{attribute 'GeneratedUsingTerminal: EK1122-0000-0018'}
{attribute addProperty BoxType "EK1122-0000-0018"}
{attribute addProperty Id "Beckhoff_EPP3xxxsub_EK1100EK1100_1FC0878B2A_0001_EPP3174_0002_0016EPP3174_DCC7866252A_0002_EPP3174_0002_0017EPP3174_DCC7866252A_0003_EPP3174_0002_0018EPP3174_DCC7866252A_0004_EPP3184_0002_0016EPP3184_DCC7866252A_0005_EPP3184_0002_0017EPP3184_DCC7866252A_0006_EPP3184_0002_0018EPP3184_DCC7866252A_0007_EPP3184_0002_0019EPP3184_DCC7866252A_0008_EPP3204_0002_0016EPP3204_6CD7E11952A_0009_EPP3204_0002_0017EPP3204_5380707048A_0010_EPP3204_0002_0018EPP3204_5380707048A_0011_EPP3204_0002_0019EPP3204_5380707048A_0012_EPP3314_0002_0016EPP3314_B654D23048A_0013_EPP3314_0002_0017EPP3314_B654D23048A_0014_EPP3314_0002_0018EPP3314_B654D23048A_0015_EPP3632_0001_0016EPP3632_E2B98A5C86A_0016_EPP3632_0001_0017EPP3632_E2B98A5C86A_0017_EPP3744_0041_0016EPP3744_315C92D470A_0018_EPP3744_0041_0017EPP3744_315C92D470A_0019_EPP3744_0041_0018EPP3744_315C92D470A_0020_EPP3744_1041_0016EPP3744_315C92D470A_0021_EPP3744_1041_0017EPP3744_315C92D470A_0022_EPP3744_1041_0018EPP3744_315C92D470A_0023_EPP3744_1041_0019EPP3744_315C92D470A_0024_EPP3744_1041_0020EPP3744_315C92D470A_0025_EPP3752_0000_0017EPP3752_C992DA1B42"}
{attribute addProperty CRC "2576063294"}
{attribute addProperty Size "1480"}
TYPE Beckhoff_EPP3xxxEK1122_998B9B3E EXTENDS EK1122_1FC0878B :
STRUCT
	{attribute addProperty Name "Beckhoff_EPP3xxxsub_EK1100"}
	{attribute addProperty PreviousPort "Beckhoff EPP3xxxEK1122 : D"}
	Beckhoff_EPP3xxxsub_EK1100 : EK1100_1FC0878B;
	{attribute addProperty Name "A_0001_EPP3174_0002_0016"}
	{attribute addProperty PreviousPort "Beckhoff EPP3xxxsub EK1100 : C"}
	A_0001_EPP3174_0002_0016 : EPP3174_DCC78662;
	{attribute addProperty Name "A_0002_EPP3174_0002_0017"}
	{attribute addProperty PreviousPort "A_0001(EPP3174-0002-0016) : B"}
	A_0002_EPP3174_0002_0017 : EPP3174_DCC78662;
	{attribute addProperty Name "A_0003_EPP3174_0002_0018"}
	{attribute addProperty PreviousPort "A_0002(EPP3174-0002-0017) : B"}
	A_0003_EPP3174_0002_0018 : EPP3174_DCC78662;
	{attribute addProperty Name "A_0004_EPP3184_0002_0016"}
	{attribute addProperty PreviousPort "A_0003(EPP3174-0002-0018) : B"}
	A_0004_EPP3184_0002_0016 : EPP3184_DCC78662;
	{attribute addProperty Name "A_0005_EPP3184_0002_0017"}
	{attribute addProperty PreviousPort "A_0004(EPP3184-0002-0016) : B"}
	A_0005_EPP3184_0002_0017 : EPP3184_DCC78662;
	{attribute addProperty Name "A_0006_EPP3184_0002_0018"}
	{attribute addProperty PreviousPort "A_0005(EPP3184-0002-0017) : B"}
	A_0006_EPP3184_0002_0018 : EPP3184_DCC78662;
	{attribute addProperty Name "A_0007_EPP3184_0002_0019"}
	{attribute addProperty PreviousPort "A_0006(EPP3184-0002-0018) : B"}
	A_0007_EPP3184_0002_0019 : EPP3184_DCC78662;
	{attribute addProperty Name "A_0008_EPP3204_0002_0016"}
	{attribute addProperty PreviousPort "A_0007(EPP3184-0002-0019) : B"}
	A_0008_EPP3204_0002_0016 : EPP3204_6CD7E119;
	{attribute addProperty Name "A_0009_EPP3204_0002_0017"}
	{attribute addProperty PreviousPort "A_0008(EPP3204-0002-0016) : B"}
	A_0009_EPP3204_0002_0017 : EPP3204_53807070;
	{attribute addProperty Name "A_0010_EPP3204_0002_0018"}
	{attribute addProperty PreviousPort "A_0009(EPP3204-0002-0017) : B"}
	A_0010_EPP3204_0002_0018 : EPP3204_53807070;
	{attribute addProperty Name "A_0011_EPP3204_0002_0019"}
	{attribute addProperty PreviousPort "A_0010(EPP3204-0002-0018) : B"}
	A_0011_EPP3204_0002_0019 : EPP3204_53807070;
	{attribute addProperty Name "A_0012_EPP3314_0002_0016"}
	{attribute addProperty PreviousPort "A_0011(EPP3204-0002-0019) : B"}
	A_0012_EPP3314_0002_0016 : EPP3314_B654D230;
	{attribute addProperty Name "A_0013_EPP3314_0002_0017"}
	{attribute addProperty PreviousPort "A_0012(EPP3314-0002-0016) : B"}
	A_0013_EPP3314_0002_0017 : EPP3314_B654D230;
	{attribute addProperty Name "A_0014_EPP3314_0002_0018"}
	{attribute addProperty PreviousPort "A_0013(EPP3314-0002-0017) : B"}
	A_0014_EPP3314_0002_0018 : EPP3314_B654D230;
	{attribute addProperty Name "A_0015_EPP3632_0001_0016"}
	{attribute addProperty PreviousPort "A_0014(EPP3314-0002-0018) : B"}
	A_0015_EPP3632_0001_0016 : EPP3632_E2B98A5C;
	{attribute addProperty Name "A_0016_EPP3632_0001_0017"}
	{attribute addProperty PreviousPort "A_0015(EPP3632-0001-0016) : B"}
	A_0016_EPP3632_0001_0017 : EPP3632_E2B98A5C;
	{attribute addProperty Name "A_0017_EPP3744_0041_0016"}
	{attribute addProperty PreviousPort "A_0016(EPP3632-0001-0017) : B"}
	A_0017_EPP3744_0041_0016 : EPP3744_315C92D4;
	{attribute addProperty Name "A_0018_EPP3744_0041_0017"}
	{attribute addProperty PreviousPort "A_0017(EPP3744-0041-0016) : B"}
	A_0018_EPP3744_0041_0017 : EPP3744_315C92D4;
	{attribute addProperty Name "A_0019_EPP3744_0041_0018"}
	{attribute addProperty PreviousPort "A_0018(EPP3744-0041-0017) : B"}
	A_0019_EPP3744_0041_0018 : EPP3744_315C92D4;
	{attribute addProperty Name "A_0020_EPP3744_1041_0016"}
	{attribute addProperty PreviousPort "A_0019(EPP3744-0041-0018) : B"}
	A_0020_EPP3744_1041_0016 : EPP3744_315C92D4;
	{attribute addProperty Name "A_0021_EPP3744_1041_0017"}
	{attribute addProperty PreviousPort "A_0020(EPP3744-1041-0016) : B"}
	A_0021_EPP3744_1041_0017 : EPP3744_315C92D4;
	{attribute addProperty Name "A_0022_EPP3744_1041_0018"}
	{attribute addProperty PreviousPort "A_0021(EPP3744-1041-0017) : B"}
	A_0022_EPP3744_1041_0018 : EPP3744_315C92D4;
	{attribute addProperty Name "A_0023_EPP3744_1041_0019"}
	{attribute addProperty PreviousPort "A_0022(EPP3744-1041-0018) : B"}
	A_0023_EPP3744_1041_0019 : EPP3744_315C92D4;
	{attribute addProperty Name "A_0024_EPP3744_1041_0020"}
	{attribute addProperty PreviousPort "A_0023(EPP3744-1041-0019) : B"}
	A_0024_EPP3744_1041_0020 : EPP3744_315C92D4;
	{attribute addProperty Name "A_0025_EPP3752_0000_0017"}
	{attribute addProperty PreviousPort "A_0024(EPP3744-1041-0020) : B"}
	A_0025_EPP3752_0000_0017 : EPP3752_C992DA1B;
END_STRUCT
END_TYPE

(* stored: Version 1.2.0.0, ProductVersion 3.1.4024.9
   DUT Beckhoff_EPP3xxxEK1122_998B9B3E: Id {31ae6827-803a-4192-97d2-ad4f597fb9d9} *)
